TYPE Waypoint :
	STRUCT
		x, y : LREAL;
	 	mode: PointMode; 		// 1 = docking, 2 = transfer, -1 = datenpunkt nicht verwendet
	END_STRUCT
END_TYPE

(* stored: Version 1.1.0.1, ProductVersion 3.1.4024.11
   DUT Waypoint: Id {e465bc3a-2c48-4cc5-85c0-ef919ef44d25} *)
